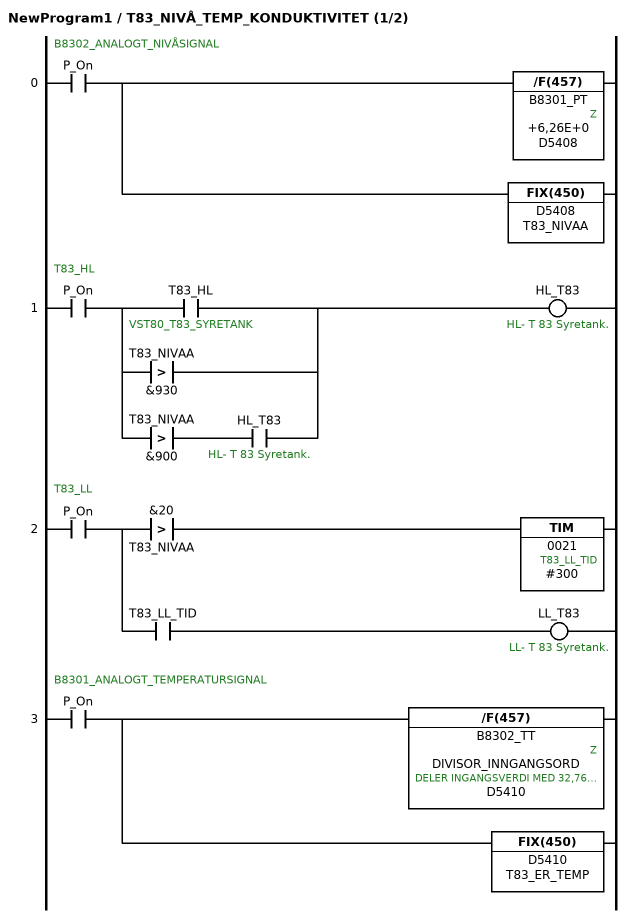
; [picture p48: NewProgram1 / T83_NIVÅ_TEMP_KONDUKTIVITET, rungs 0-3]
; rung 0: B8302_ANALOGT_NIVÅSIGNAL
LD P_On
/F(457) B8301_PT +6,26E+0 D5408  ; Z
FIX(450) D5408 T83_NIVAA
; rung 1: T83_HL
LD P_On
LD T83_HL  ; VST80_T83_SYRETANK
OR>(320) T83_NIVAA &930
LD>(320) T83_NIVAA &900
AND HL_T83  ; HL- T 83 Syretank.
ORLD
ANDLD
OUT HL_T83  ; HL- T 83 Syretank.
; rung 2: T83_LL
LD P_On
OUT TR0
AND>(320) &20 T83_NIVAA
TIM 0021 #300  ; T83_LL_TID
LD TR0
AND T83_LL_TID
OUT LL_T83  ; LL- T 83 Syretank.
; rung 3: B8301_ANALOGT_TEMPERATURSIGNAL
LD P_On
/F(457) B8302_TT DIVISOR_INNGANGSORD D5410  ; Z, DELER INGANGSVERDI MED 32,760 FOR OMREGNING TIL 0-1000
FIX(450) D5410 T83_ER_TEMP

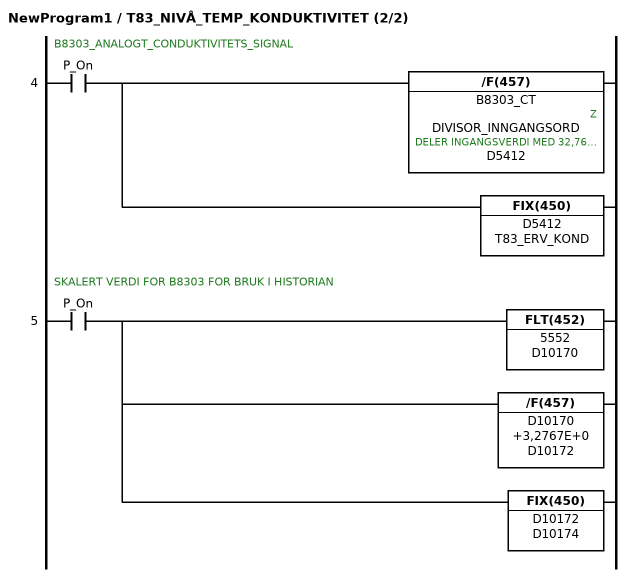
; rung 4: B8303_ANALOGT_CONDUKTIVITETS_SIGNAL
LD P_On
/F(457) B8303_CT DIVISOR_INNGANGSORD D5412  ; Z, DELER INGANGSVERDI MED 32,760 FOR OMREGNING TIL 0-1000
FIX(450) D5412 T83_ERV_KOND
; rung 5: SKALERT VERDI FOR B8303 FOR BRUK I HISTORIAN
LD P_On
FLT(452) 5552 D10170
/F(457) D10170 +3,2767E+0 D10172
FIX(450) D10172 D10174

### Section T83_FUNKSJONER_OBJEKTER

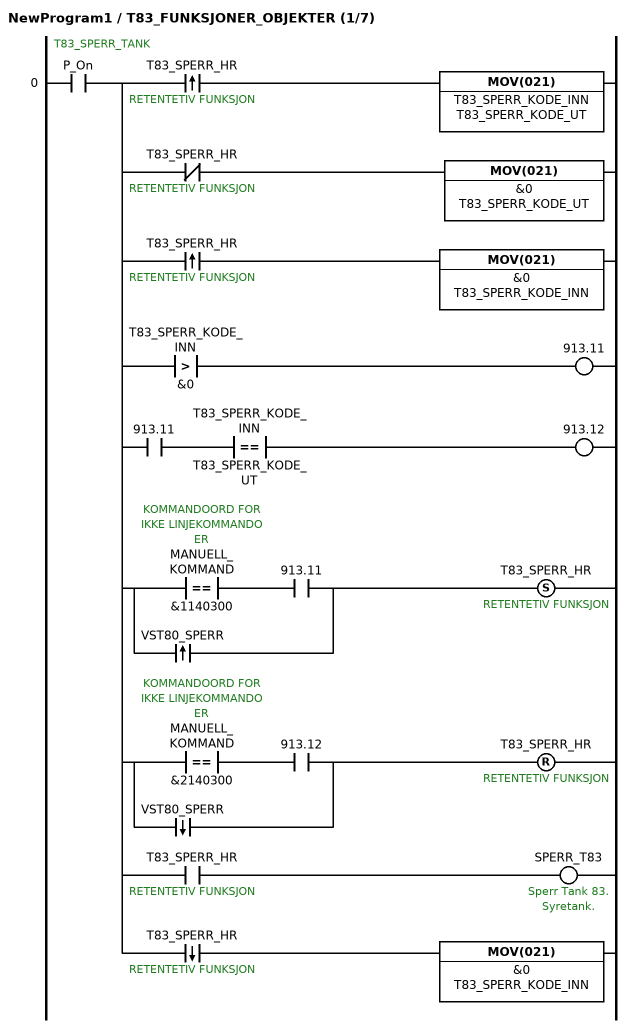
; rung 0: T83_SPERR_TANK
LD P_On
OUT TR0
@AND T83_SPERR_HR  ; RETENTETIV FUNKSJON
MOV(021) T83_SPERR_KODE_INN T83_SPERR_KODE_UT
LD TR0
ANDNOT T83_SPERR_HR  ; RETENTETIV FUNKSJON
MOV(021) &0 T83_SPERR_KODE_UT
LD TR0
@AND T83_SPERR_HR  ; RETENTETIV FUNKSJON
MOV(021) &0 T83_SPERR_KODE_INN
LD TR0
AND>(320) T83_SPERR_KODE_INN &0
OUT 913.11
LD TR0
AND 913.11
AND=(300) T83_SPERR_KODE_INN T83_SPERR_KODE_UT
OUT 913.12
LD TR0
LD=L(301) MANUELL_KOMMAND &1140300  ; KOMMANDOORD FOR IKKE LINJEKOMMANDOER
AND 913.11
@OR VST80_SPERR
ANDLD
SET T83_SPERR_HR  ; RETENTETIV FUNKSJON
LD TR0
LD=L(301) MANUELL_KOMMAND &2140300  ; KOMMANDOORD FOR IKKE LINJEKOMMANDOER
AND 913.12
%OR VST80_SPERR
ANDLD
RSET T83_SPERR_HR  ; RETENTETIV FUNKSJON
LD TR0
AND T83_SPERR_HR  ; RETENTETIV FUNKSJON
OUT SPERR_T83  ; Sperr Tank 83. Syretank.
LD TR0
%AND T83_SPERR_HR  ; RETENTETIV FUNKSJON
MOV(021) &0 T83_SPERR_KODE_INN

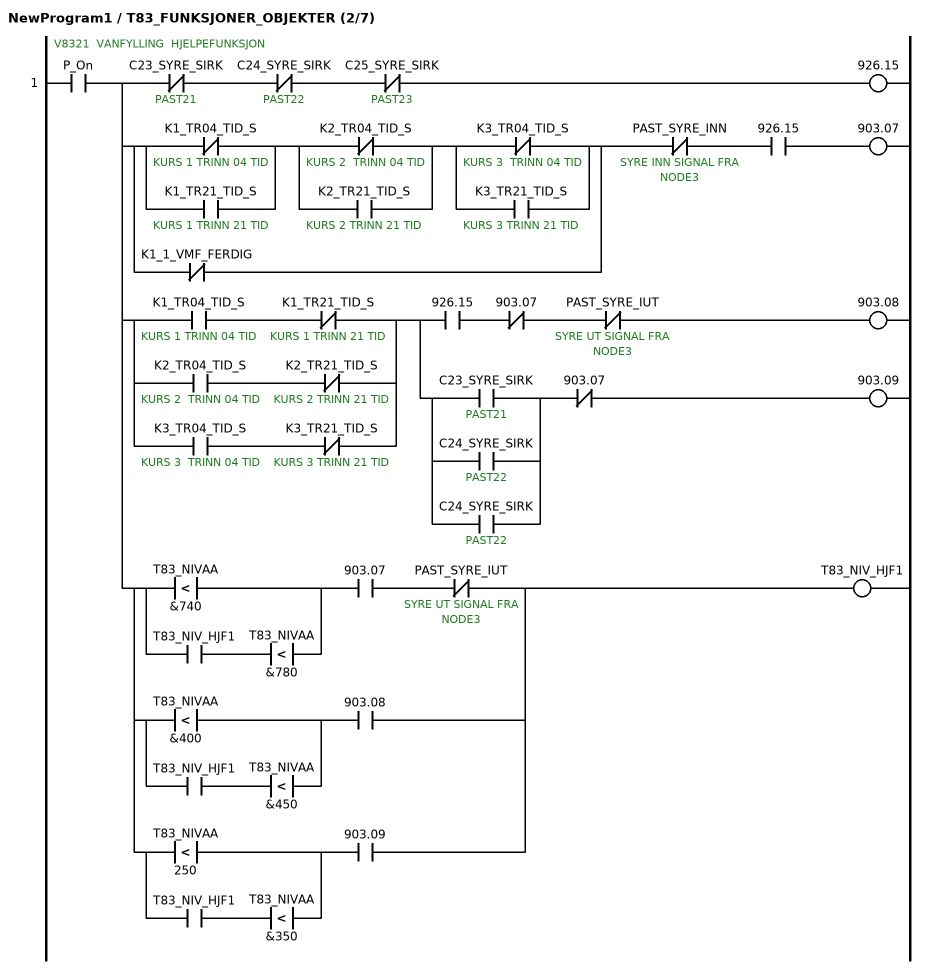
; rung 1: V8321  VANFYLLING  HJELPEFUNKSJON
LD P_On
OUT TR0
ANDNOT C23_SYRE_SIRK  ; PAST21
ANDNOT C24_SYRE_SIRK  ; PAST22
ANDNOT C25_SYRE_SIRK  ; PAST23
OUT 926.15
LD TR0
LDNOT K1_TR04_TID_S  ; KURS 1 TRINN 04 TID
OR K1_TR21_TID_S  ; KURS 1 TRINN 21 TID
LDNOT K2_TR04_TID_S  ; KURS 2  TRINN 04 TID
OR K2_TR21_TID_S  ; KURS 2 TRINN 21 TID
ANDLD
LDNOT K3_TR04_TID_S  ; KURS 3  TRINN 04 TID
OR K3_TR21_TID_S  ; KURS 3 TRINN 21 TID
ANDLD
ORNOT K1_1_VMF_FERDIG
ANDLD
ANDNOT PAST_SYRE_INN  ; SYRE INN SIGNAL FRA NODE3
AND 926.15
OUT 903.07
LD TR0
LD K1_TR04_TID_S  ; KURS 1 TRINN 04 TID
ANDNOT K1_TR21_TID_S  ; KURS 1 TRINN 21 TID
LD K2_TR04_TID_S  ; KURS 2  TRINN 04 TID
ANDNOT K2_TR21_TID_S  ; KURS 2 TRINN 21 TID
ORLD
LD K3_TR04_TID_S  ; KURS 3  TRINN 04 TID
ANDNOT K3_TR21_TID_S  ; KURS 3 TRINN 21 TID
ORLD
ANDLD
OUT TR1
AND 926.15
ANDNOT 903.07
ANDNOT PAST_SYRE_IUT  ; SYRE UT SIGNAL FRA NODE3
OUT 903.08
LD TR1
LD C23_SYRE_SIRK  ; PAST21
OR C24_SYRE_SIRK  ; PAST22
OR C24_SYRE_SIRK  ; PAST22
ANDLD
ANDNOT 903.07
OUT 903.09
LD TR0
LD<(310) T83_NIVAA &740
LD T83_NIV_HJF1
AND<(310) T83_NIVAA &780
ORLD
AND 903.07
ANDNOT PAST_SYRE_IUT  ; SYRE UT SIGNAL FRA NODE3
LD<(310) T83_NIVAA &400
LD T83_NIV_HJF1
AND<(310) T83_NIVAA &450
ORLD
AND 903.08
ORLD
LD<(310) T83_NIVAA 250
LD T83_NIV_HJF1
AND<(310) T83_NIVAA &350
ORLD
AND 903.09
ORLD
ANDLD
OUT T83_NIV_HJF1

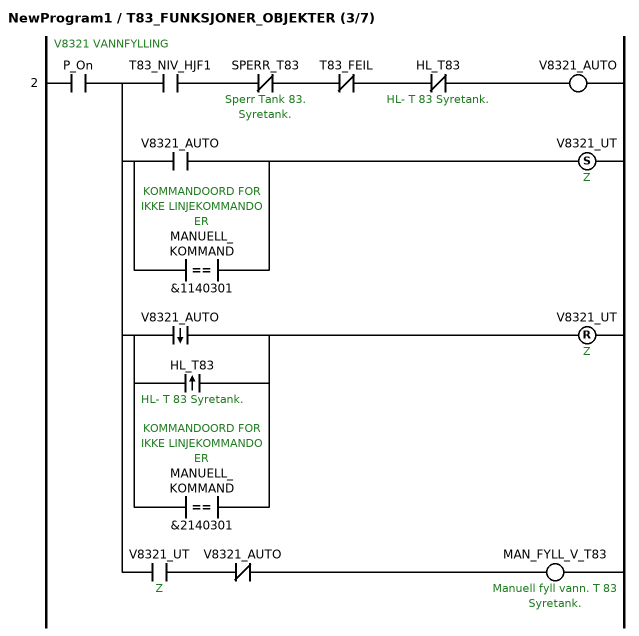
; rung 2: V8321 VANNFYLLING
LD P_On
OUT TR0
AND T83_NIV_HJF1
ANDNOT SPERR_T83  ; Sperr Tank 83. Syretank.
ANDNOT T83_FEIL
ANDNOT HL_T83  ; HL- T 83 Syretank.
OUT V8321_AUTO
LD TR0
LD V8321_AUTO
OR=L(301) MANUELL_KOMMAND &1140301  ; KOMMANDOORD FOR IKKE LINJEKOMMANDOER
ANDLD
SET V8321_UT  ; Z
LD TR0
%LD V8321_AUTO
@OR HL_T83  ; HL- T 83 Syretank.
OR=L(301) MANUELL_KOMMAND &2140301  ; KOMMANDOORD FOR IKKE LINJEKOMMANDOER
ANDLD
RSET V8321_UT  ; Z
LD TR0
AND V8321_UT  ; Z
ANDNOT V8321_AUTO
OUT MAN_FYLL_V_T83  ; Manuell fyll vann. T 83 Syretank.

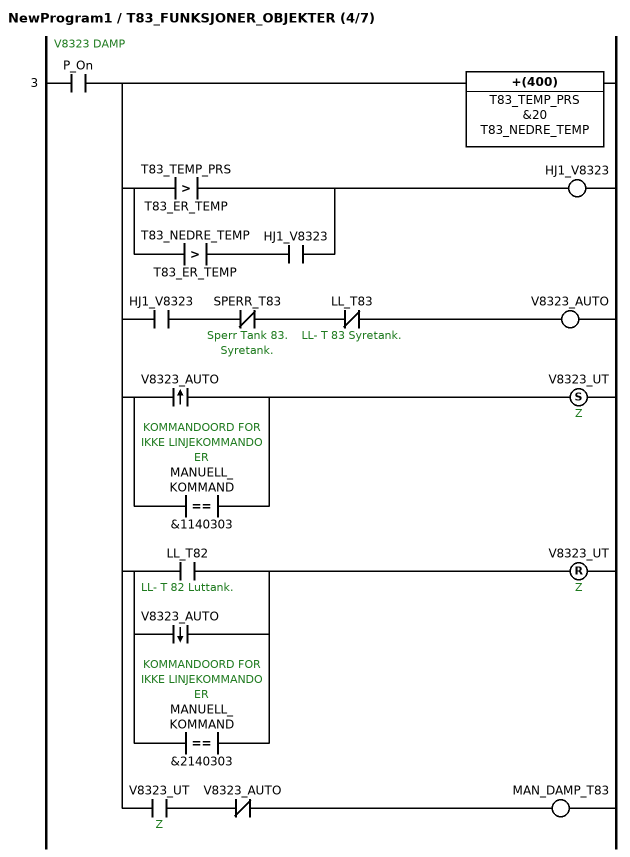
; rung 3: V8323 DAMP
LD P_On
OUT TR0
+(400) T83_TEMP_PRS &20 T83_NEDRE_TEMP
LD>(320) T83_TEMP_PRS T83_ER_TEMP
LD>(320) T83_NEDRE_TEMP T83_ER_TEMP
AND HJ1_V8323
ORLD
ANDLD
OUT HJ1_V8323
LD TR0
AND HJ1_V8323
ANDNOT SPERR_T83  ; Sperr Tank 83. Syretank.
ANDNOT LL_T83  ; LL- T 83 Syretank.
OUT V8323_AUTO
LD TR0
@LD V8323_AUTO
OR=L(301) MANUELL_KOMMAND &1140303  ; KOMMANDOORD FOR IKKE LINJEKOMMANDOER
ANDLD
SET V8323_UT  ; Z
LD TR0
LD LL_T82  ; LL- T 82 Luttank.
%OR V8323_AUTO
OR=L(301) MANUELL_KOMMAND &2140303  ; KOMMANDOORD FOR IKKE LINJEKOMMANDOER
ANDLD
RSET V8323_UT  ; Z
LD TR0
AND V8323_UT  ; Z
ANDNOT V8323_AUTO
OUT MAN_DAMP_T83

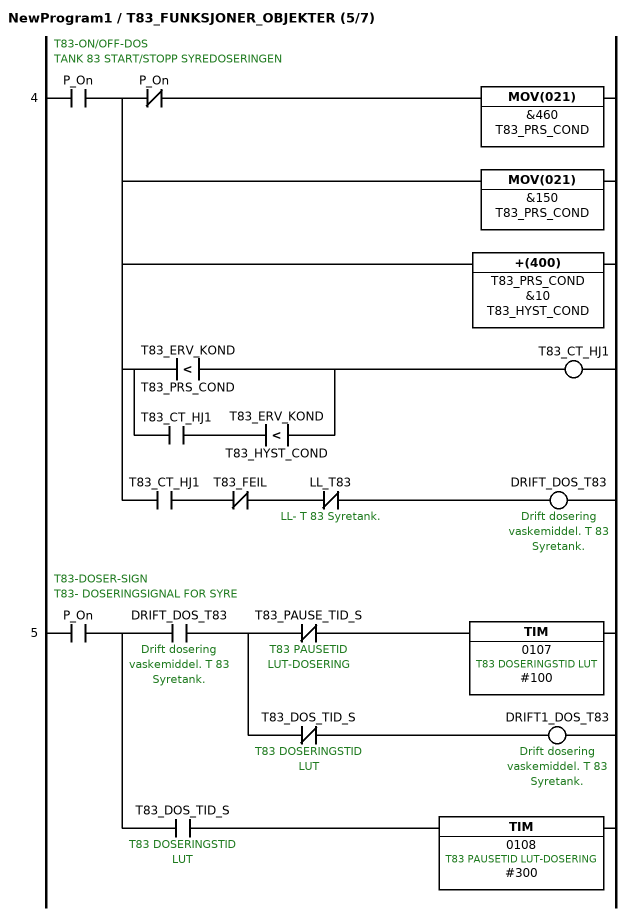
; rung 4: T83-ON/OFF-DOS / TANK 83 START/STOPP SYREDOSERINGEN
LD P_On
OUT TR0
ANDNOT P_On
MOV(021) &460 T83_PRS_COND
LD TR0
MOV(021) &150 T83_PRS_COND
+(400) T83_PRS_COND &10 T83_HYST_COND
LD<(310) T83_ERV_KOND T83_PRS_COND
LD T83_CT_HJ1
AND<(310) T83_ERV_KOND T83_HYST_COND
ORLD
ANDLD
OUT T83_CT_HJ1
LD TR0
AND T83_CT_HJ1
ANDNOT T83_FEIL
ANDNOT LL_T83  ; LL- T 83 Syretank.
OUT DRIFT_DOS_T83  ; Drift dosering vaskemiddel. T 83 Syretank.
; rung 5: T83-DOSER-SIGN / T83- DOSERINGSIGNAL FOR SYRE
LD P_On
OUT TR0
AND DRIFT_DOS_T83  ; Drift dosering vaskemiddel. T 83 Syretank.
OUT TR1
ANDNOT T83_PAUSE_TID_S  ; T83 PAUSETID LUT-DOSERING
TIM 0107 #100  ; T83 DOSERINGSTID LUT
LD TR1
ANDNOT T83_DOS_TID_S  ; T83 DOSERINGSTID LUT
OUT DRIFT1_DOS_T83  ; Drift dosering vaskemiddel. T 83 Syretank.
LD TR0
AND T83_DOS_TID_S  ; T83 DOSERINGSTID LUT
TIM 0108 #300  ; T83 PAUSETID LUT-DOSERING

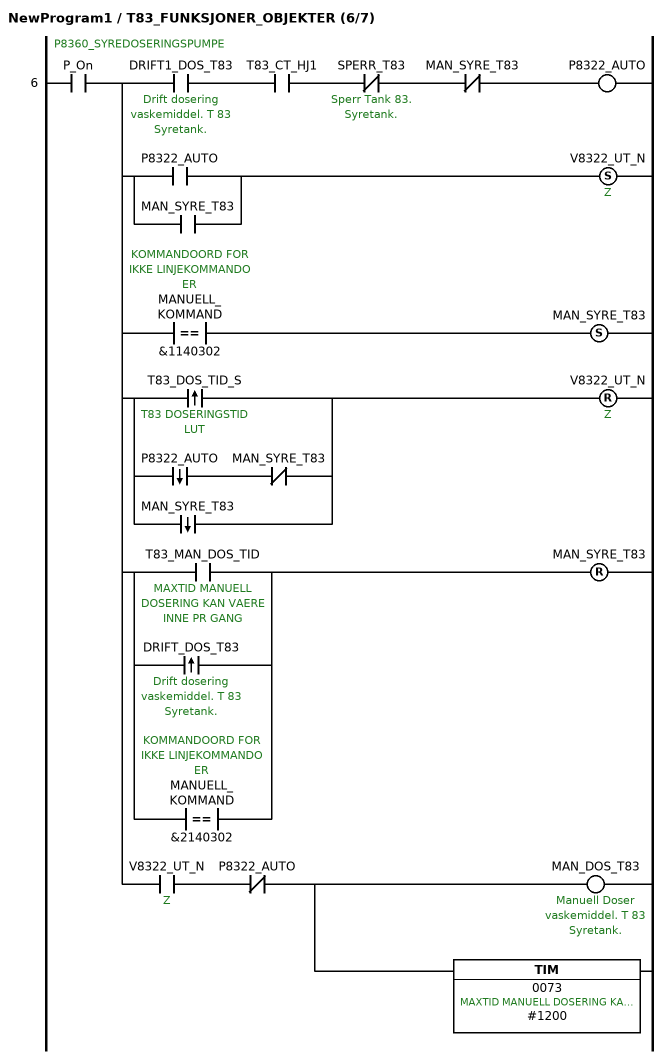
; rung 6: P8360_SYREDOSERINGSPUMPE
LD P_On
OUT TR0
AND DRIFT1_DOS_T83  ; Drift dosering vaskemiddel. T 83 Syretank.
AND T83_CT_HJ1
ANDNOT SPERR_T83  ; Sperr Tank 83. Syretank.
ANDNOT MAN_SYRE_T83
OUT P8322_AUTO
LD TR0
LD P8322_AUTO
OR MAN_SYRE_T83
ANDLD
SET V8322_UT_N  ; Z
LD TR0
AND=L(301) MANUELL_KOMMAND &1140302  ; KOMMANDOORD FOR IKKE LINJEKOMMANDOER
SET MAN_SYRE_T83
LD TR0
@LD T83_DOS_TID_S  ; T83 DOSERINGSTID LUT
%LD P8322_AUTO
ANDNOT MAN_SYRE_T83
ORLD
%OR MAN_SYRE_T83
ANDLD
RSET V8322_UT_N  ; Z
LD TR0
LD T83_MAN_DOS_TID  ; MAXTID MANUELL DOSERING KAN VAERE INNE PR GANG
@OR DRIFT_DOS_T83  ; Drift dosering vaskemiddel. T 83 Syretank.
OR=L(301) MANUELL_KOMMAND &2140302  ; KOMMANDOORD FOR IKKE LINJEKOMMANDOER
ANDLD
RSET MAN_SYRE_T83
LD TR0
AND V8322_UT_N  ; Z
ANDNOT P8322_AUTO
OUT MAN_DOS_T83  ; Manuell Doser vaskemiddel. T 83 Syretank.
TIM 0073 #1200  ; MAXTID MANUELL DOSERING KAN VAERE INNE PR GANG

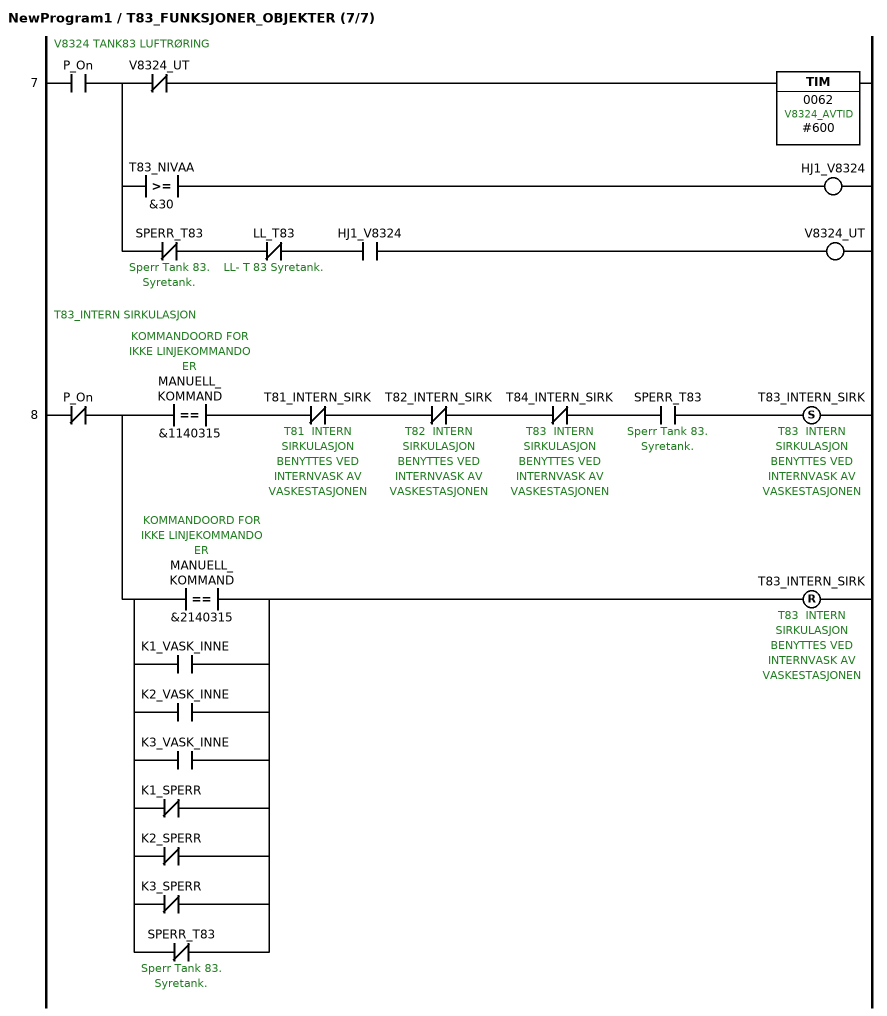
; rung 7: V8324 TANK83 LUFTRØRING
LD P_On
OUT TR0
ANDNOT V8324_UT
TIM 0062 #600  ; V8324_AVTID
LD TR0
AND>=(325) T83_NIVAA &30
OUT HJ1_V8324
LD TR0
ANDNOT SPERR_T83  ; Sperr Tank 83. Syretank.
ANDNOT LL_T83  ; LL- T 83 Syretank.
AND HJ1_V8324
OUT V8324_UT
; rung 8: T83_INTERN SIRKULASJON
LDNOT P_On
OUT TR0
AND=L(301) MANUELL_KOMMAND &1140315  ; KOMMANDOORD FOR IKKE LINJEKOMMANDOER
ANDNOT T81_INTERN_SIRK  ; T81  INTERN SIRKULASJON BENYTTES VED INTERNVASK AV VASKESTASJONEN
ANDNOT T82_INTERN_SIRK  ; T82  INTERN SIRKULASJON BENYTTES VED INTERNVASK AV VASKESTASJONEN
ANDNOT T84_INTERN_SIRK  ; T83  INTERN SIRKULASJON BENYTTES VED INTERNVASK AV VASKESTASJONEN
AND SPERR_T83  ; Sperr Tank 83. Syretank.
SET T83_INTERN_SIRK  ; T83  INTERN SIRKULASJON BENYTTES VED INTERNVASK AV VASKESTASJONEN
LD TR0
LD=L(301) MANUELL_KOMMAND &2140315  ; KOMMANDOORD FOR IKKE LINJEKOMMANDOER
OR K1_VASK_INNE
OR K2_VASK_INNE
OR K3_VASK_INNE
ORNOT K1_SPERR
ORNOT K2_SPERR
ORNOT K3_SPERR
ORNOT SPERR_T83  ; Sperr Tank 83. Syretank.
ANDLD
RSET T83_INTERN_SIRK  ; T83  INTERN SIRKULASJON BENYTTES VED INTERNVASK AV VASKESTASJONEN

### Section T84_NIVÅ_TEMPERATUR_CONDUKTIVITET

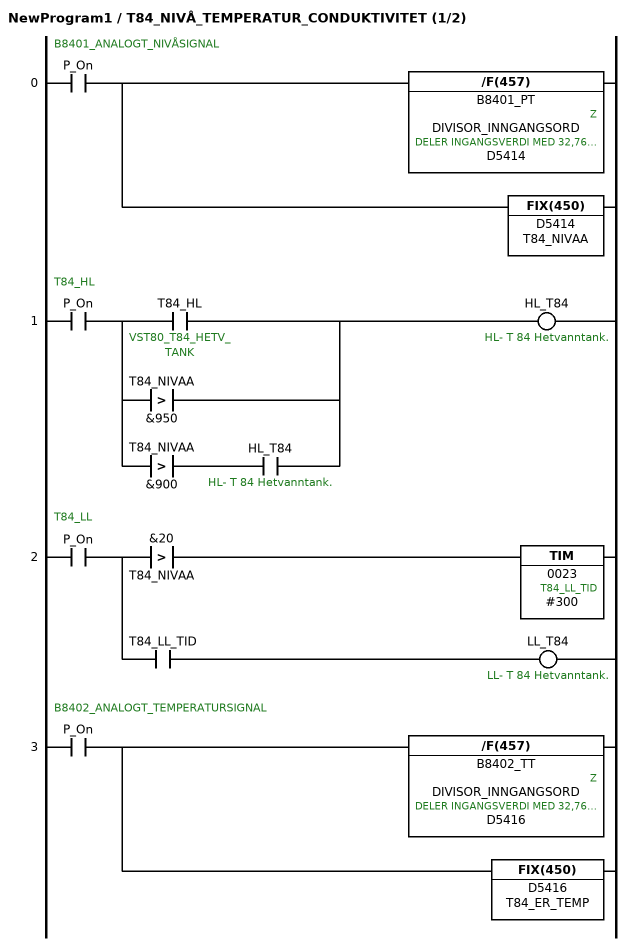
; rung 0: B8401_ANALOGT_NIVÅSIGNAL
LD P_On
/F(457) B8401_PT DIVISOR_INNGANGSORD D5414  ; Z, DELER INGANGSVERDI MED 32,760 FOR OMREGNING TIL 0-1000
FIX(450) D5414 T84_NIVAA
; rung 1: T84_HL
LD P_On
LD T84_HL  ; VST80_T84_HETV_TANK
OR>(320) T84_NIVAA &950
LD>(320) T84_NIVAA &900
AND HL_T84  ; HL- T 84 Hetvanntank.
ORLD
ANDLD
OUT HL_T84  ; HL- T 84 Hetvanntank.
; rung 2: T84_LL
LD P_On
OUT TR0
AND>(320) &20 T84_NIVAA
TIM 0023 #300  ; T84_LL_TID
LD TR0
AND T84_LL_TID
OUT LL_T84  ; LL- T 84 Hetvanntank.
; rung 3: B8402_ANALOGT_TEMPERATURSIGNAL
LD P_On
/F(457) B8402_TT DIVISOR_INNGANGSORD D5416  ; Z, DELER INGANGSVERDI MED 32,760 FOR OMREGNING TIL 0-1000
FIX(450) D5416 T84_ER_TEMP

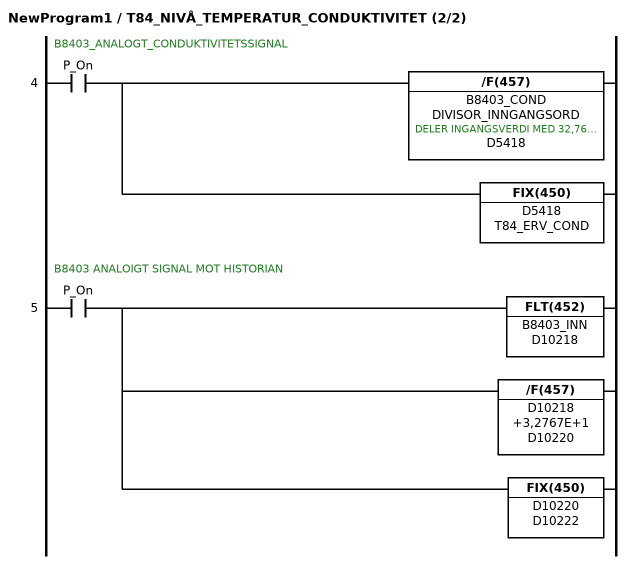
; rung 4: B8403_ANALOGT_CONDUKTIVITETSSIGNAL
LD P_On
/F(457) B8403_COND DIVISOR_INNGANGSORD D5418  ; DELER INGANGSVERDI MED 32,760 FOR OMREGNING TIL 0-1000
FIX(450) D5418 T84_ERV_COND
; rung 5: B8403 ANALOIGT SIGNAL MOT HISTORIAN
LD P_On
FLT(452) B8403_INN D10218
/F(457) D10218 +3,2767E+1 D10220
FIX(450) D10220 D10222

### Section T84_FUNKSJONER_OBJEKTER

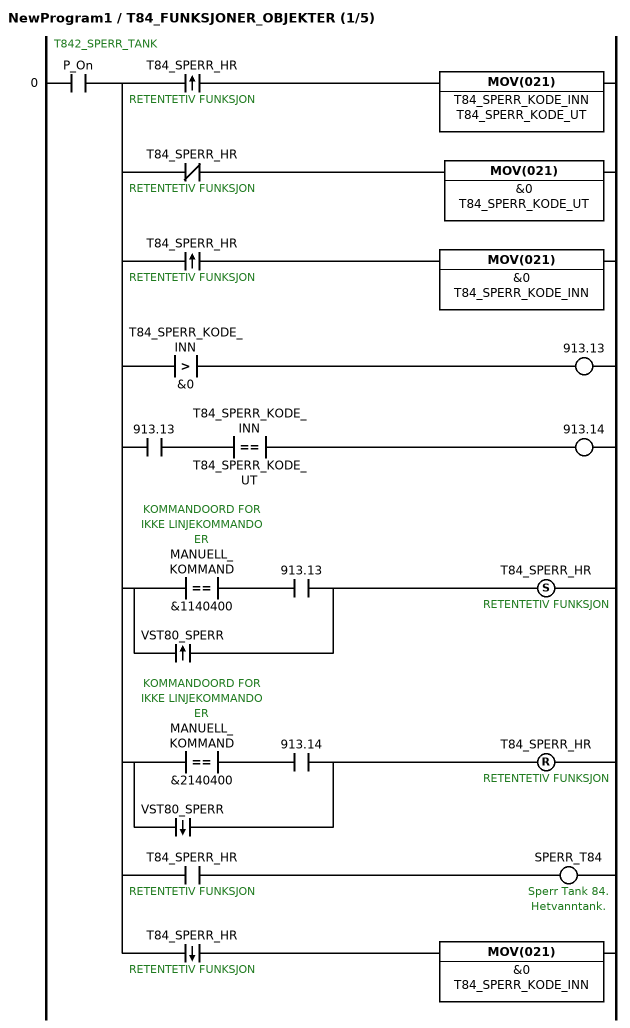
; rung 0: T842_SPERR_TANK
LD P_On
OUT TR0
@AND T84_SPERR_HR  ; RETENTETIV FUNKSJON
MOV(021) T84_SPERR_KODE_INN T84_SPERR_KODE_UT
LD TR0
ANDNOT T84_SPERR_HR  ; RETENTETIV FUNKSJON
MOV(021) &0 T84_SPERR_KODE_UT
LD TR0
@AND T84_SPERR_HR  ; RETENTETIV FUNKSJON
MOV(021) &0 T84_SPERR_KODE_INN
LD TR0
AND>(320) T84_SPERR_KODE_INN &0
OUT 913.13
LD TR0
AND 913.13
AND=(300) T84_SPERR_KODE_INN T84_SPERR_KODE_UT
OUT 913.14
LD TR0
LD=L(301) MANUELL_KOMMAND &1140400  ; KOMMANDOORD FOR IKKE LINJEKOMMANDOER
AND 913.13
@OR VST80_SPERR
ANDLD
SET T84_SPERR_HR  ; RETENTETIV FUNKSJON
LD TR0
LD=L(301) MANUELL_KOMMAND &2140400  ; KOMMANDOORD FOR IKKE LINJEKOMMANDOER
AND 913.14
%OR VST80_SPERR
ANDLD
RSET T84_SPERR_HR  ; RETENTETIV FUNKSJON
LD TR0
AND T84_SPERR_HR  ; RETENTETIV FUNKSJON
OUT SPERR_T84  ; Sperr Tank 84. Hetvanntank.
LD TR0
%AND T84_SPERR_HR  ; RETENTETIV FUNKSJON
MOV(021) &0 T84_SPERR_KODE_INN

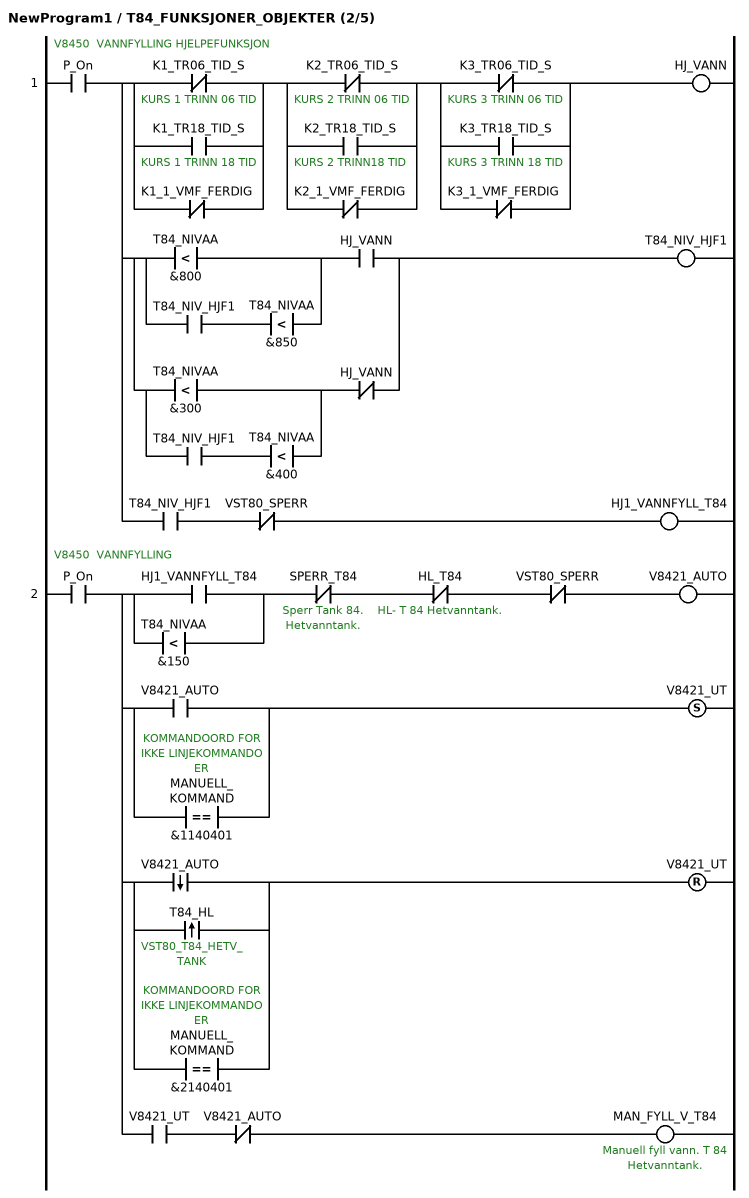
; rung 1: V8450  VANNFYLLING HJELPEFUNKSJON
LD P_On
OUT TR0
LDNOT K1_TR06_TID_S  ; KURS 1 TRINN 06 TID
OR K1_TR18_TID_S  ; KURS 1 TRINN 18 TID
ORNOT K1_1_VMF_FERDIG
ANDLD
LDNOT K2_TR06_TID_S  ; KURS 2 TRINN 06 TID
OR K2_TR18_TID_S  ; KURS 2 TRINN18 TID
ORNOT K2_1_VMF_FERDIG
ANDLD
LDNOT K3_TR06_TID_S  ; KURS 3 TRINN 06 TID
OR K3_TR18_TID_S  ; KURS 3 TRINN 18 TID
ORNOT K3_1_VMF_FERDIG
ANDLD
OUT HJ_VANN
LD TR0
LD<(310) T84_NIVAA &800
LD T84_NIV_HJF1
AND<(310) T84_NIVAA &850
ORLD
AND HJ_VANN
LD<(310) T84_NIVAA &300
LD T84_NIV_HJF1
AND<(310) T84_NIVAA &400
ORLD
ANDNOT HJ_VANN
ORLD
ANDLD
OUT T84_NIV_HJF1
LD TR0
AND T84_NIV_HJF1
ANDNOT VST80_SPERR
OUT HJ1_VANNFYLL_T84
; rung 2: V8450  VANNFYLLING
LD P_On
OUT TR0
LD HJ1_VANNFYLL_T84
OR<(310) T84_NIVAA &150
ANDLD
ANDNOT SPERR_T84  ; Sperr Tank 84. Hetvanntank.
ANDNOT HL_T84  ; HL- T 84 Hetvanntank.
ANDNOT VST80_SPERR
OUT V8421_AUTO
LD TR0
LD V8421_AUTO
OR=L(301) MANUELL_KOMMAND &1140401  ; KOMMANDOORD FOR IKKE LINJEKOMMANDOER
ANDLD
SET V8421_UT
LD TR0
%LD V8421_AUTO
@OR T84_HL  ; VST80_T84_HETV_TANK
OR=L(301) MANUELL_KOMMAND &2140401  ; KOMMANDOORD FOR IKKE LINJEKOMMANDOER
ANDLD
RSET V8421_UT
LD TR0
AND V8421_UT
ANDNOT V8421_AUTO
OUT MAN_FYLL_V_T84  ; Manuell fyll vann. T 84 Hetvanntank.

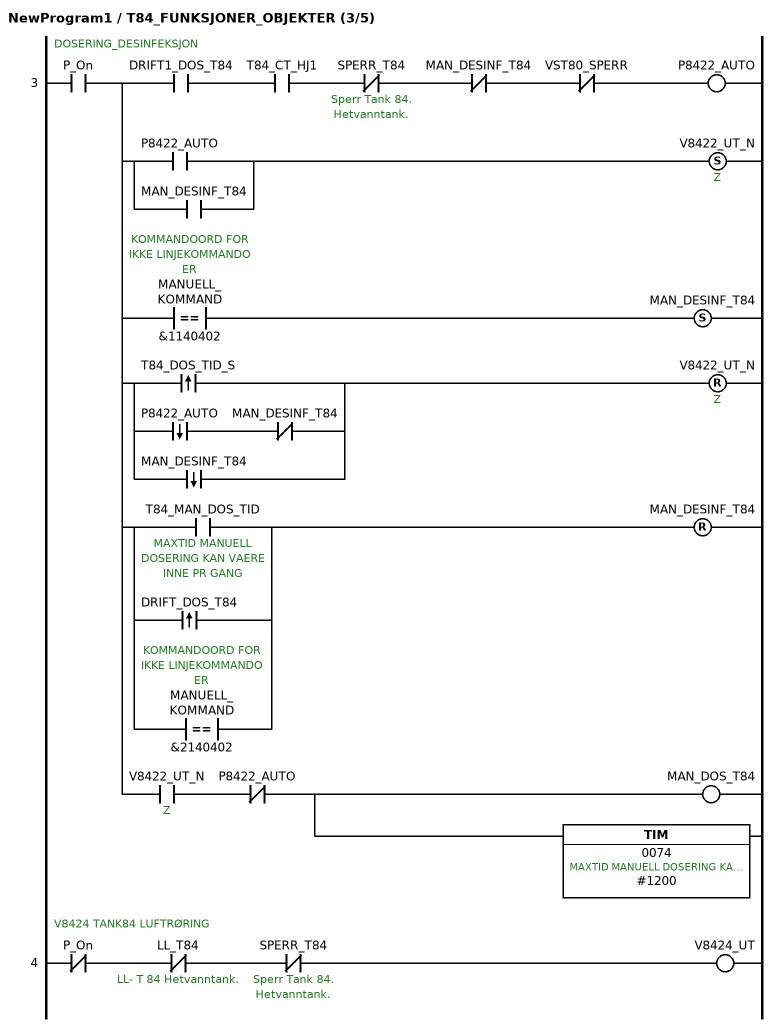
; rung 3: DOSERING_DESINFEKSJON
LD P_On
OUT TR0
AND DRIFT1_DOS_T84
AND T84_CT_HJ1
ANDNOT SPERR_T84  ; Sperr Tank 84. Hetvanntank.
ANDNOT MAN_DESINF_T84
ANDNOT VST80_SPERR
OUT P8422_AUTO
LD TR0
LD P8422_AUTO
OR MAN_DESINF_T84
ANDLD
SET V8422_UT_N  ; Z
LD TR0
AND=L(301) MANUELL_KOMMAND &1140402  ; KOMMANDOORD FOR IKKE LINJEKOMMANDOER
SET MAN_DESINF_T84
LD TR0
@LD T84_DOS_TID_S
%LD P8422_AUTO
ANDNOT MAN_DESINF_T84
ORLD
%OR MAN_DESINF_T84
ANDLD
RSET V8422_UT_N  ; Z
LD TR0
LD T84_MAN_DOS_TID  ; MAXTID MANUELL DOSERING KAN VAERE INNE PR GANG
@OR DRIFT_DOS_T84
OR=L(301) MANUELL_KOMMAND &2140402  ; KOMMANDOORD FOR IKKE LINJEKOMMANDOER
ANDLD
RSET MAN_DESINF_T84
LD TR0
AND V8422_UT_N  ; Z
ANDNOT P8422_AUTO
OUT MAN_DOS_T84
TIM 0074 #1200  ; MAXTID MANUELL DOSERING KAN VAERE INNE PR GANG
; rung 4: V8424 TANK84 LUFTRØRING
LDNOT P_On
ANDNOT LL_T84  ; LL- T 84 Hetvanntank.
ANDNOT SPERR_T84  ; Sperr Tank 84. Hetvanntank.
OUT V8424_UT

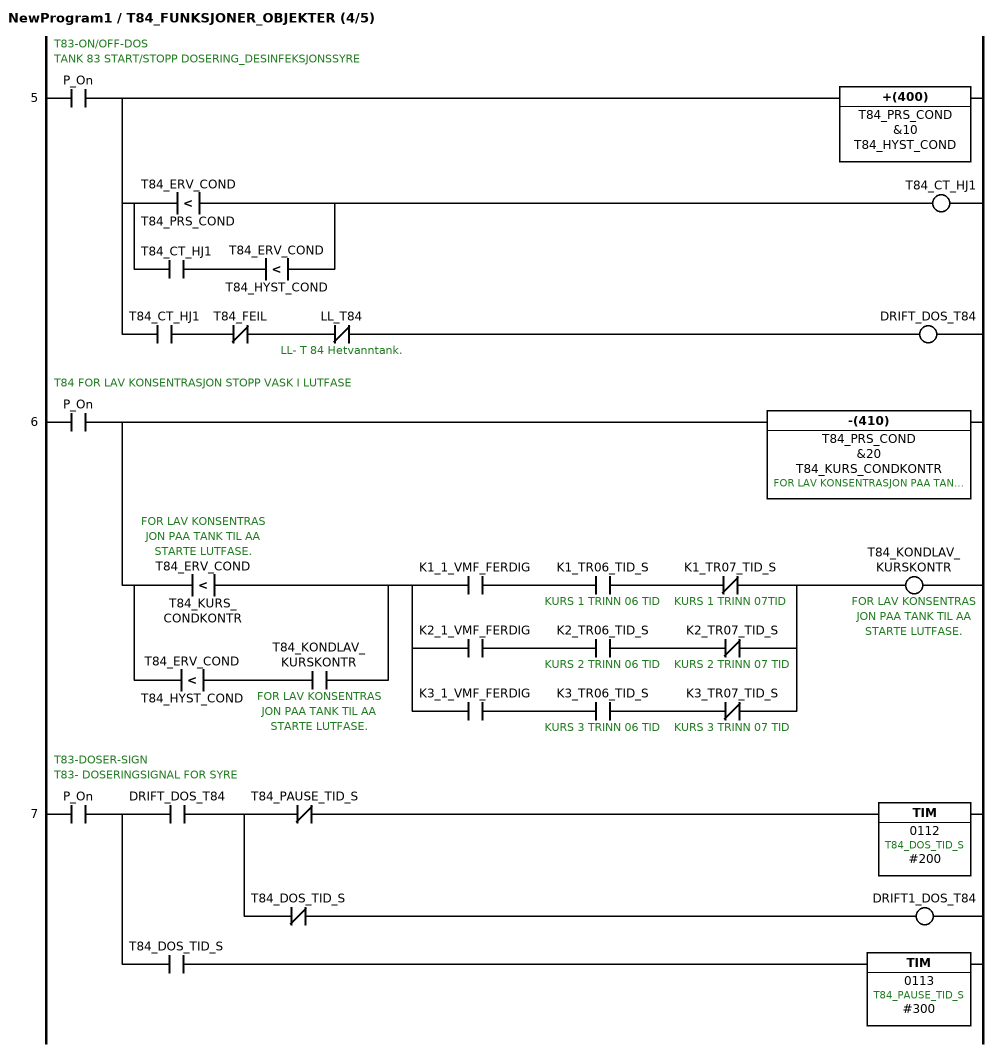
; rung 5: T83-ON/OFF-DOS / TANK 83 START/STOPP DOSERING_DESINFEKSJONSSYRE
LD P_On
OUT TR0
+(400) T84_PRS_COND &10 T84_HYST_COND
LD<(310) T84_ERV_COND T84_PRS_COND
LD T84_CT_HJ1
AND<(310) T84_ERV_COND T84_HYST_COND
ORLD
ANDLD
OUT T84_CT_HJ1
LD TR0
AND T84_CT_HJ1
ANDNOT T84_FEIL
ANDNOT LL_T84  ; LL- T 84 Hetvanntank.
OUT DRIFT_DOS_T84
; rung 6: T84 FOR LAV KONSENTRASJON STOPP VASK I LUTFASE
LD P_On
-(410) T84_PRS_COND &20 T84_KURS_CONDKONTR  ; FOR LAV KONSENTRASJON PAA TANK TIL AA STARTE LUTFASE.
LD<(310) T84_ERV_COND T84_KURS_CONDKONTR  ; FOR LAV KONSENTRASJON PAA TANK TIL AA STARTE LUTFASE.
LD<(310) T84_ERV_COND T84_HYST_COND
AND T84_KONDLAV_KURSKONTR  ; FOR LAV KONSENTRASJON PAA TANK TIL AA STARTE LUTFASE.
ORLD
ANDLD
LD K1_1_VMF_FERDIG
AND K1_TR06_TID_S  ; KURS 1 TRINN 06 TID
ANDNOT K1_TR07_TID_S  ; KURS 1 TRINN 07TID
LD K2_1_VMF_FERDIG
AND K2_TR06_TID_S  ; KURS 2 TRINN 06 TID
ANDNOT K2_TR07_TID_S  ; KURS 2 TRINN 07 TID
ORLD
LD K3_1_VMF_FERDIG
AND K3_TR06_TID_S  ; KURS 3 TRINN 06 TID
ANDNOT K3_TR07_TID_S  ; KURS 3 TRINN 07 TID
ORLD
ANDLD
OUT T84_KONDLAV_KURSKONTR  ; FOR LAV KONSENTRASJON PAA TANK TIL AA STARTE LUTFASE.
; rung 7: T83-DOSER-SIGN / T83- DOSERINGSIGNAL FOR SYRE
LD P_On
OUT TR0
AND DRIFT_DOS_T84
OUT TR1
ANDNOT T84_PAUSE_TID_S
TIM 0112 #200  ; T84_DOS_TID_S
LD TR1
ANDNOT T84_DOS_TID_S
OUT DRIFT1_DOS_T84
LD TR0
AND T84_DOS_TID_S
TIM 0113 #300  ; T84_PAUSE_TID_S

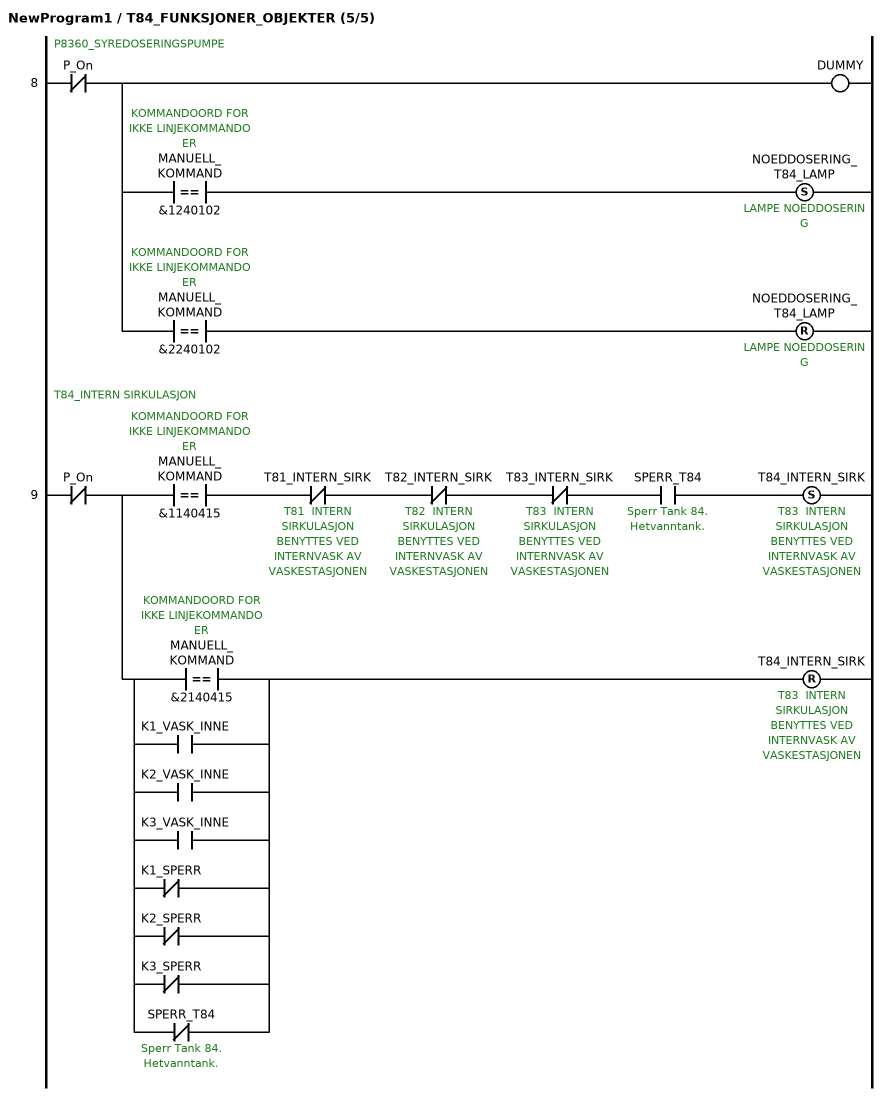
; rung 8: P8360_SYREDOSERINGSPUMPE
LDNOT P_On
OUT TR0
OUT DUMMY
AND=L(301) MANUELL_KOMMAND &1240102  ; KOMMANDOORD FOR IKKE LINJEKOMMANDOER
SET NOEDDOSERING_T84_LAMP  ; LAMPE NOEDDOSERING
LD TR0
AND=L(301) MANUELL_KOMMAND &2240102  ; KOMMANDOORD FOR IKKE LINJEKOMMANDOER
RSET NOEDDOSERING_T84_LAMP  ; LAMPE NOEDDOSERING
; rung 9: T84_INTERN SIRKULASJON
LDNOT P_On
OUT TR0
AND=L(301) MANUELL_KOMMAND &1140415  ; KOMMANDOORD FOR IKKE LINJEKOMMANDOER
ANDNOT T81_INTERN_SIRK  ; T81  INTERN SIRKULASJON BENYTTES VED INTERNVASK AV VASKESTASJONEN
ANDNOT T82_INTERN_SIRK  ; T82  INTERN SIRKULASJON BENYTTES VED INTERNVASK AV VASKESTASJONEN
ANDNOT T83_INTERN_SIRK  ; T83  INTERN SIRKULASJON BENYTTES VED INTERNVASK AV VASKESTASJONEN
AND SPERR_T84  ; Sperr Tank 84. Hetvanntank.
SET T84_INTERN_SIRK  ; T83  INTERN SIRKULASJON BENYTTES VED INTERNVASK AV VASKESTASJONEN
LD TR0
LD=L(301) MANUELL_KOMMAND &2140415  ; KOMMANDOORD FOR IKKE LINJEKOMMANDOER
OR K1_VASK_INNE
OR K2_VASK_INNE
OR K3_VASK_INNE
ORNOT K1_SPERR
ORNOT K2_SPERR
ORNOT K3_SPERR
ORNOT SPERR_T84  ; Sperr Tank 84. Hetvanntank.
ANDLD
RSET T84_INTERN_SIRK  ; T83  INTERN SIRKULASJON BENYTTES VED INTERNVASK AV VASKESTASJONEN

### Section VST80_TANKFEIL

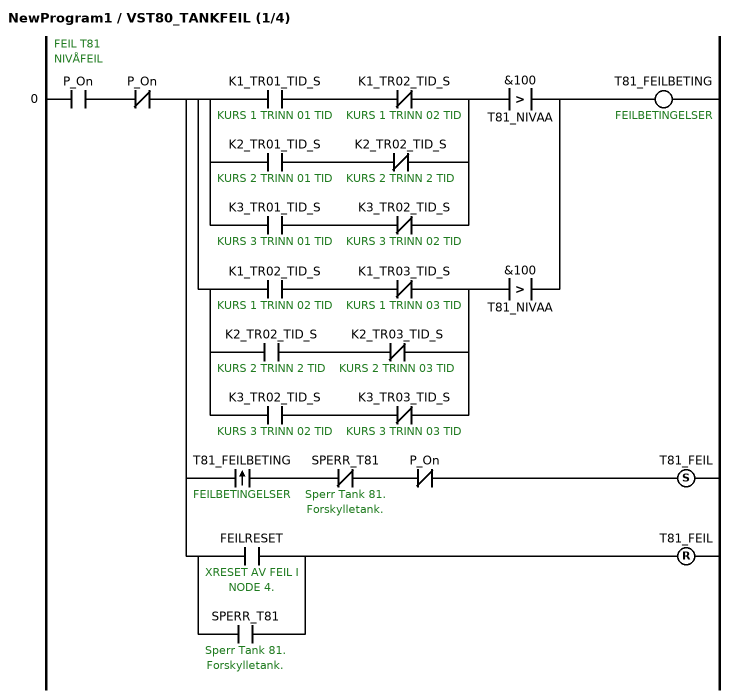
; rung 0: FEIL T81 / NIVÅFEIL
LD P_On
ANDNOT P_On
OUT TR0
LD K1_TR01_TID_S  ; KURS 1 TRINN 01 TID
ANDNOT K1_TR02_TID_S  ; KURS 1 TRINN 02 TID
LD K2_TR01_TID_S  ; KURS 2 TRINN 01 TID
ANDNOT K2_TR02_TID_S  ; KURS 2 TRINN 2 TID
ORLD
LD K3_TR01_TID_S  ; KURS 3 TRINN 01 TID
ANDNOT K3_TR02_TID_S  ; KURS 3 TRINN 02 TID
ORLD
AND>(320) &100 T81_NIVAA
LD K1_TR02_TID_S  ; KURS 1 TRINN 02 TID
ANDNOT K1_TR03_TID_S  ; KURS 1 TRINN 03 TID
LD K2_TR02_TID_S  ; KURS 2 TRINN 2 TID
ANDNOT K2_TR03_TID_S  ; KURS 2 TRINN 03 TID
ORLD
LD K3_TR02_TID_S  ; KURS 3 TRINN 02 TID
ANDNOT K3_TR03_TID_S  ; KURS 3 TRINN 03 TID
ORLD
AND>(320) &100 T81_NIVAA
ORLD
ANDLD
OUT T81_FEILBETING  ; FEILBETINGELSER
LD TR0
@AND T81_FEILBETING  ; FEILBETINGELSER
ANDNOT SPERR_T81  ; Sperr Tank 81. Forskylletank.
ANDNOT P_On
SET T81_FEIL
LD TR0
LD FEILRESET  ; XRESET AV FEIL I NODE 4.
OR SPERR_T81  ; Sperr Tank 81. Forskylletank.
ANDLD
RSET T81_FEIL

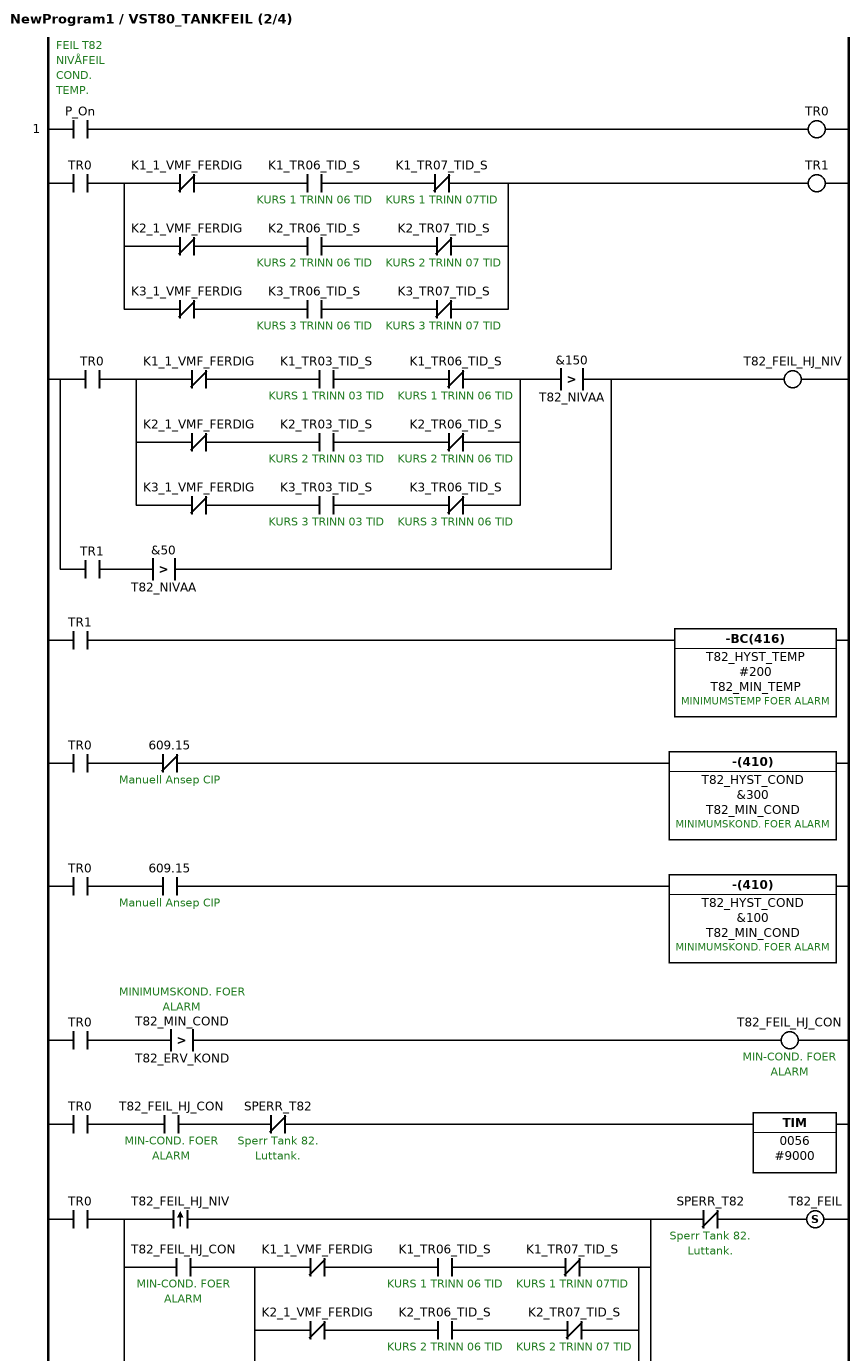

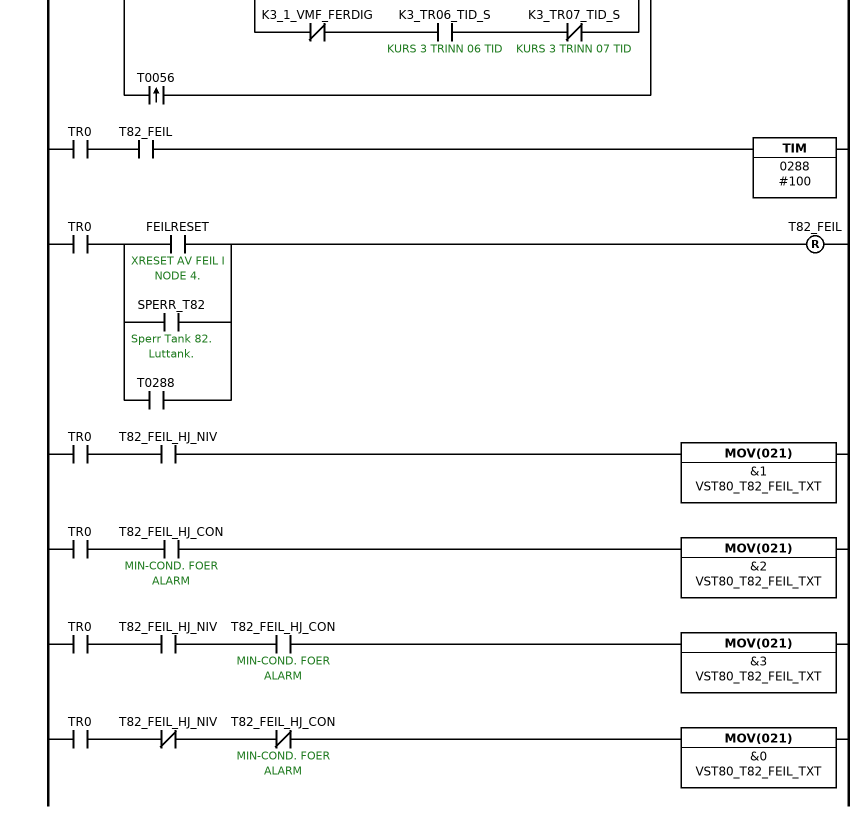
; rung 1: FEIL T82 / NIVÅFEIL / COND. / TEMP.
LD P_On
OUT TR0
LDNOT K1_1_VMF_FERDIG
AND K1_TR03_TID_S  ; KURS 1 TRINN 03 TID
ANDNOT K1_TR06_TID_S  ; KURS 1 TRINN 06 TID
LDNOT K2_1_VMF_FERDIG
AND K2_TR03_TID_S  ; KURS 2 TRINN 03 TID
ANDNOT K2_TR06_TID_S  ; KURS 2 TRINN 06 TID
ORLD
LDNOT K3_1_VMF_FERDIG
AND K3_TR03_TID_S  ; KURS 3 TRINN 03 TID
ANDNOT K3_TR06_TID_S  ; KURS 3 TRINN 06 TID
ORLD
ANDLD
AND>(320) &150 T82_NIVAA
LD TR0
LDNOT K1_1_VMF_FERDIG
AND K1_TR06_TID_S  ; KURS 1 TRINN 06 TID
ANDNOT K1_TR07_TID_S  ; KURS 1 TRINN 07TID
LDNOT K2_1_VMF_FERDIG
AND K2_TR06_TID_S  ; KURS 2 TRINN 06 TID
ANDNOT K2_TR07_TID_S  ; KURS 2 TRINN 07 TID
ORLD
LDNOT K3_1_VMF_FERDIG
AND K3_TR06_TID_S  ; KURS 3 TRINN 06 TID
ANDNOT K3_TR07_TID_S  ; KURS 3 TRINN 07 TID
ORLD
ANDLD
OUT TR1
AND>(320) &50 T82_NIVAA
ORLD
OUT T82_FEIL_HJ_NIV
LD TR1
-BC(416) T82_HYST_TEMP #200 T82_MIN_TEMP  ; MINIMUMSTEMP FOER ALARM
LD TR0
ANDNOT 609.15  ; Manuell Ansep CIP
-(410) T82_HYST_COND &300 T82_MIN_COND  ; MINIMUMSKOND. FOER ALARM
LD TR0
AND 609.15  ; Manuell Ansep CIP
-(410) T82_HYST_COND &100 T82_MIN_COND  ; MINIMUMSKOND. FOER ALARM
LD TR0
AND>(320) T82_MIN_COND T82_ERV_KOND  ; MINIMUMSKOND. FOER ALARM
OUT T82_FEIL_HJ_CON  ; MIN-COND. FOER ALARM
LD TR0
AND T82_FEIL_HJ_CON  ; MIN-COND. FOER ALARM
ANDNOT SPERR_T82  ; Sperr Tank 82. Luttank.
TIM 0056 #9000
LD TR0
@LD T82_FEIL_HJ_NIV
LD T82_FEIL_HJ_CON  ; MIN-COND. FOER ALARM
LDNOT K1_1_VMF_FERDIG
AND K1_TR06_TID_S  ; KURS 1 TRINN 06 TID
ANDNOT K1_TR07_TID_S  ; KURS 1 TRINN 07TID
LDNOT K2_1_VMF_FERDIG
AND K2_TR06_TID_S  ; KURS 2 TRINN 06 TID
ANDNOT K2_TR07_TID_S  ; KURS 2 TRINN 07 TID
ORLD
LDNOT K3_1_VMF_FERDIG
AND K3_TR06_TID_S  ; KURS 3 TRINN 06 TID
ANDNOT K3_TR07_TID_S  ; KURS 3 TRINN 07 TID
ORLD
ANDLD
ORLD
@OR T0056
ANDLD
ANDNOT SPERR_T82  ; Sperr Tank 82. Luttank.
SET T82_FEIL
LD TR0
AND T82_FEIL
TIM 0288 #100
LD TR0
LD FEILRESET  ; XRESET AV FEIL I NODE 4.
OR SPERR_T82  ; Sperr Tank 82. Luttank.
OR T0288
ANDLD
RSET T82_FEIL
LD TR0
AND T82_FEIL_HJ_NIV
MOV(021) &1 VST80_T82_FEIL_TXT
LD TR0
AND T82_FEIL_HJ_CON  ; MIN-COND. FOER ALARM
MOV(021) &2 VST80_T82_FEIL_TXT
LD TR0
AND T82_FEIL_HJ_NIV
AND T82_FEIL_HJ_CON  ; MIN-COND. FOER ALARM
MOV(021) &3 VST80_T82_FEIL_TXT
LD TR0
ANDNOT T82_FEIL_HJ_NIV
ANDNOT T82_FEIL_HJ_CON  ; MIN-COND. FOER ALARM
MOV(021) &0 VST80_T82_FEIL_TXT

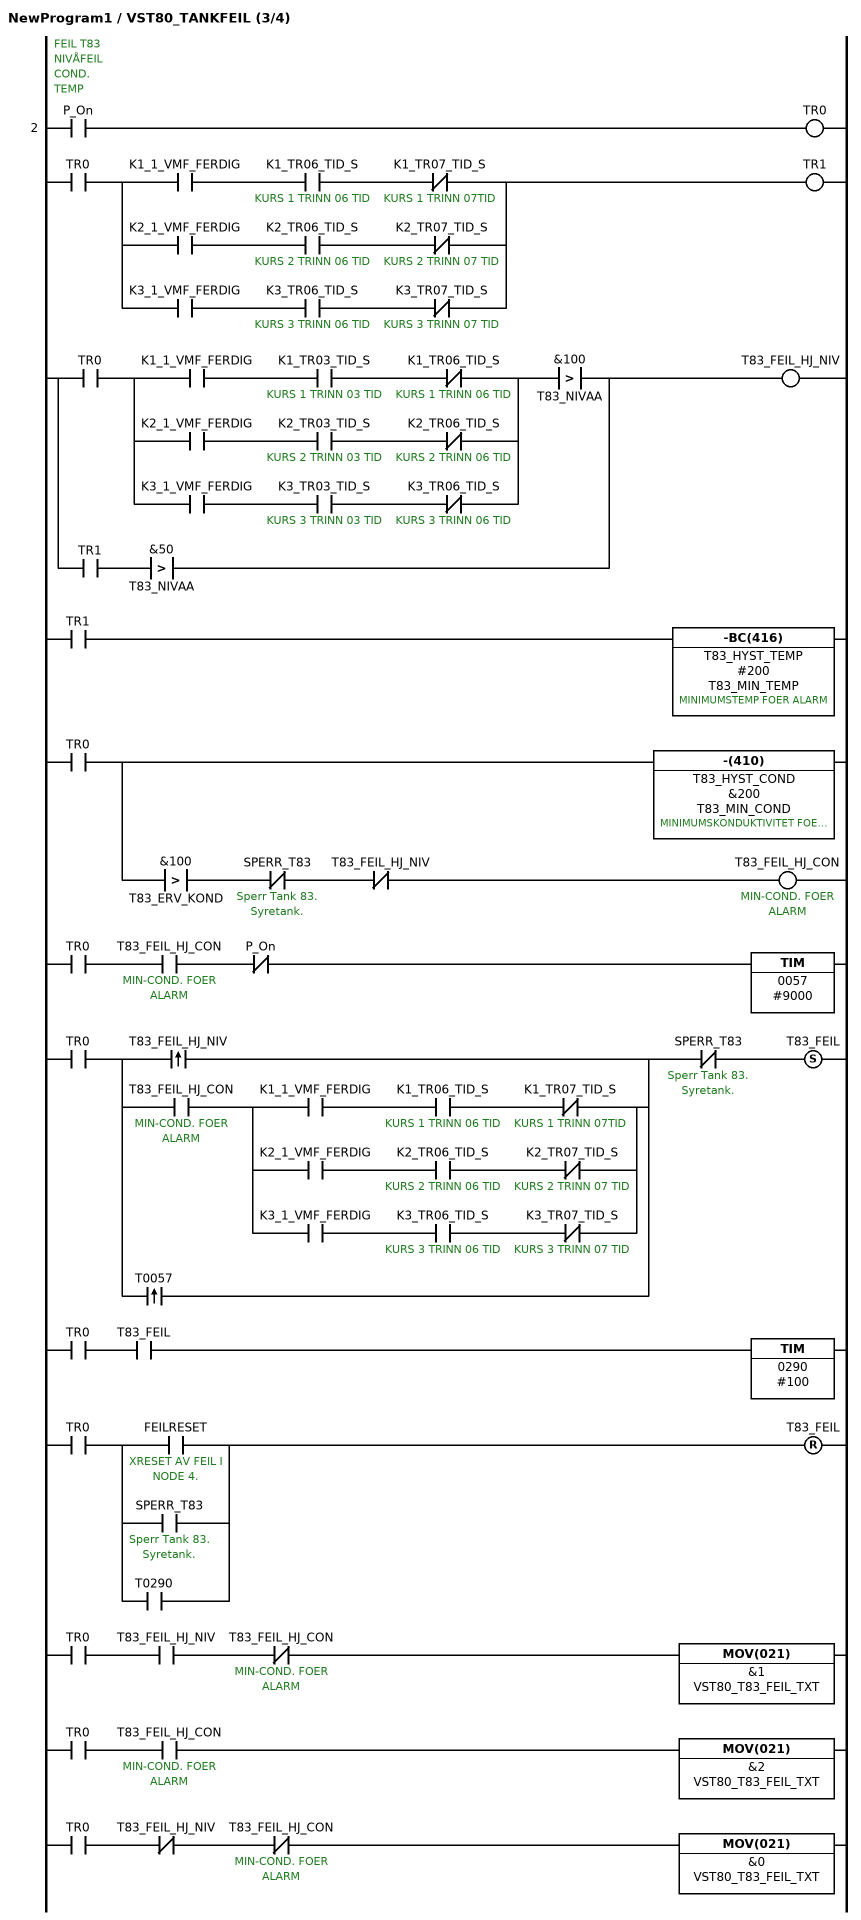
; rung 2: FEIL T83 / NIVÅFEIL / COND. / TEMP
LD P_On
OUT TR0
LD K1_1_VMF_FERDIG
AND K1_TR03_TID_S  ; KURS 1 TRINN 03 TID
ANDNOT K1_TR06_TID_S  ; KURS 1 TRINN 06 TID
LD K2_1_VMF_FERDIG
AND K2_TR03_TID_S  ; KURS 2 TRINN 03 TID
ANDNOT K2_TR06_TID_S  ; KURS 2 TRINN 06 TID
ORLD
LD K3_1_VMF_FERDIG
AND K3_TR03_TID_S  ; KURS 3 TRINN 03 TID
ANDNOT K3_TR06_TID_S  ; KURS 3 TRINN 06 TID
ORLD
ANDLD
AND>(320) &100 T83_NIVAA
LD TR0
LD K1_1_VMF_FERDIG
AND K1_TR06_TID_S  ; KURS 1 TRINN 06 TID
ANDNOT K1_TR07_TID_S  ; KURS 1 TRINN 07TID
LD K2_1_VMF_FERDIG
AND K2_TR06_TID_S  ; KURS 2 TRINN 06 TID
ANDNOT K2_TR07_TID_S  ; KURS 2 TRINN 07 TID
ORLD
LD K3_1_VMF_FERDIG
AND K3_TR06_TID_S  ; KURS 3 TRINN 06 TID
ANDNOT K3_TR07_TID_S  ; KURS 3 TRINN 07 TID
ORLD
ANDLD
OUT TR1
AND>(320) &50 T83_NIVAA
ORLD
OUT T83_FEIL_HJ_NIV
LD TR1
-BC(416) T83_HYST_TEMP #200 T83_MIN_TEMP  ; MINIMUMSTEMP FOER ALARM
LD TR0
-(410) T83_HYST_COND &200 T83_MIN_COND  ; MINIMUMSKONDUKTIVITET FOER ALARM
AND>(320) &100 T83_ERV_KOND
ANDNOT SPERR_T83  ; Sperr Tank 83. Syretank.
ANDNOT T83_FEIL_HJ_NIV
OUT T83_FEIL_HJ_CON  ; MIN-COND. FOER ALARM
LD TR0
AND T83_FEIL_HJ_CON  ; MIN-COND. FOER ALARM
ANDNOT P_On
TIM 0057 #9000
LD TR0
@LD T83_FEIL_HJ_NIV
LD T83_FEIL_HJ_CON  ; MIN-COND. FOER ALARM
LD K1_1_VMF_FERDIG
AND K1_TR06_TID_S  ; KURS 1 TRINN 06 TID
ANDNOT K1_TR07_TID_S  ; KURS 1 TRINN 07TID
LD K2_1_VMF_FERDIG
AND K2_TR06_TID_S  ; KURS 2 TRINN 06 TID
ANDNOT K2_TR07_TID_S  ; KURS 2 TRINN 07 TID
ORLD
LD K3_1_VMF_FERDIG
AND K3_TR06_TID_S  ; KURS 3 TRINN 06 TID
ANDNOT K3_TR07_TID_S  ; KURS 3 TRINN 07 TID
ORLD
ANDLD
ORLD
@OR T0057
ANDLD
ANDNOT SPERR_T83  ; Sperr Tank 83. Syretank.
SET T83_FEIL
LD TR0
AND T83_FEIL
TIM 0290 #100
LD TR0
LD FEILRESET  ; XRESET AV FEIL I NODE 4.
OR SPERR_T83  ; Sperr Tank 83. Syretank.
OR T0290
ANDLD
RSET T83_FEIL
LD TR0
AND T83_FEIL_HJ_NIV
ANDNOT T83_FEIL_HJ_CON  ; MIN-COND. FOER ALARM
MOV(021) &1 VST80_T83_FEIL_TXT
LD TR0
AND T83_FEIL_HJ_CON  ; MIN-COND. FOER ALARM
MOV(021) &2 VST80_T83_FEIL_TXT
LD TR0
ANDNOT T83_FEIL_HJ_NIV
ANDNOT T83_FEIL_HJ_CON  ; MIN-COND. FOER ALARM
MOV(021) &0 VST80_T83_FEIL_TXT

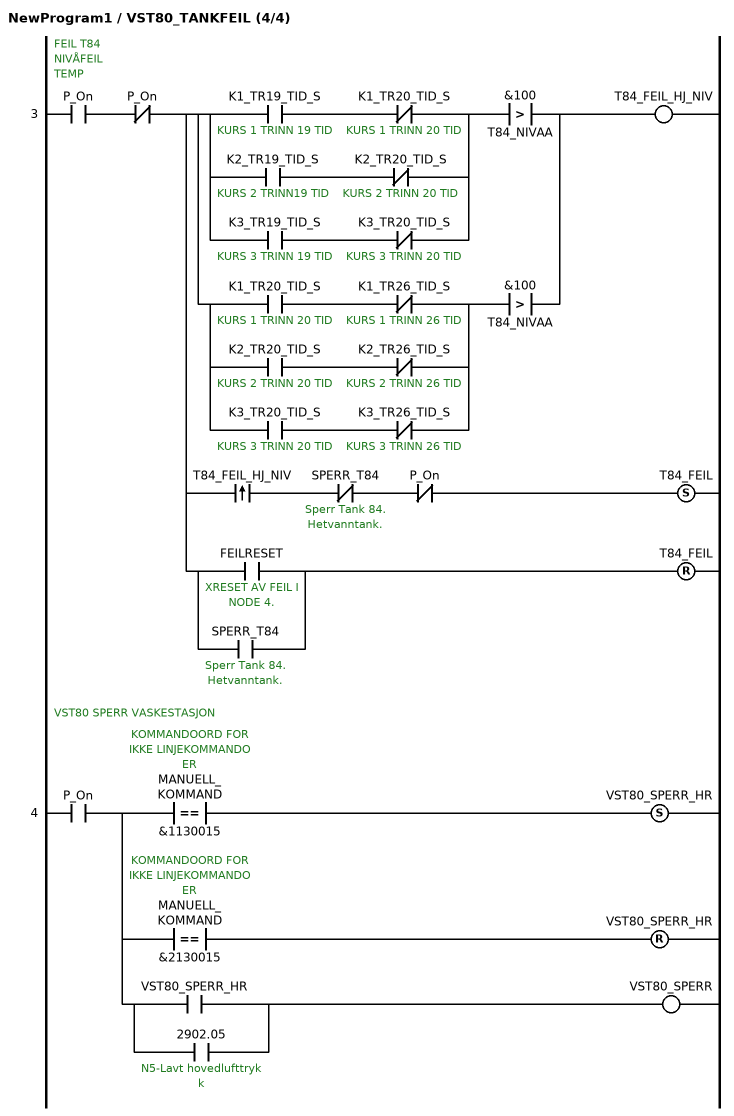
; rung 3: FEIL T84 / NIVÅFEIL / TEMP
LD P_On
ANDNOT P_On
OUT TR0
LD K1_TR19_TID_S  ; KURS 1 TRINN 19 TID
ANDNOT K1_TR20_TID_S  ; KURS 1 TRINN 20 TID
LD K2_TR19_TID_S  ; KURS 2 TRINN19 TID
ANDNOT K2_TR20_TID_S  ; KURS 2 TRINN 20 TID
ORLD
LD K3_TR19_TID_S  ; KURS 3 TRINN 19 TID
ANDNOT K3_TR20_TID_S  ; KURS 3 TRINN 20 TID
ORLD
AND>(320) &100 T84_NIVAA
LD K1_TR20_TID_S  ; KURS 1 TRINN 20 TID
ANDNOT K1_TR26_TID_S  ; KURS 1 TRINN 26 TID
LD K2_TR20_TID_S  ; KURS 2 TRINN 20 TID
ANDNOT K2_TR26_TID_S  ; KURS 2 TRINN 26 TID
ORLD
LD K3_TR20_TID_S  ; KURS 3 TRINN 20 TID
ANDNOT K3_TR26_TID_S  ; KURS 3 TRINN 26 TID
ORLD
AND>(320) &100 T84_NIVAA
ORLD
ANDLD
OUT T84_FEIL_HJ_NIV
LD TR0
@AND T84_FEIL_HJ_NIV
ANDNOT SPERR_T84  ; Sperr Tank 84. Hetvanntank.
ANDNOT P_On
SET T84_FEIL
LD TR0
LD FEILRESET  ; XRESET AV FEIL I NODE 4.
OR SPERR_T84  ; Sperr Tank 84. Hetvanntank.
ANDLD
RSET T84_FEIL
; rung 4: VST80 SPERR VASKESTASJON
LD P_On
OUT TR0
AND=L(301) MANUELL_KOMMAND &1130015  ; KOMMANDOORD FOR IKKE LINJEKOMMANDOER
SET VST80_SPERR_HR
LD TR0
AND=L(301) MANUELL_KOMMAND &2130015  ; KOMMANDOORD FOR IKKE LINJEKOMMANDOER
RSET VST80_SPERR_HR
LD TR0
LD VST80_SPERR_HR
OR 2902.05  ; N5-Lavt hovedlufttrykk
ANDLD
OUT VST80_SPERR

### Section VST80_K_1_TIDER_TR1_18

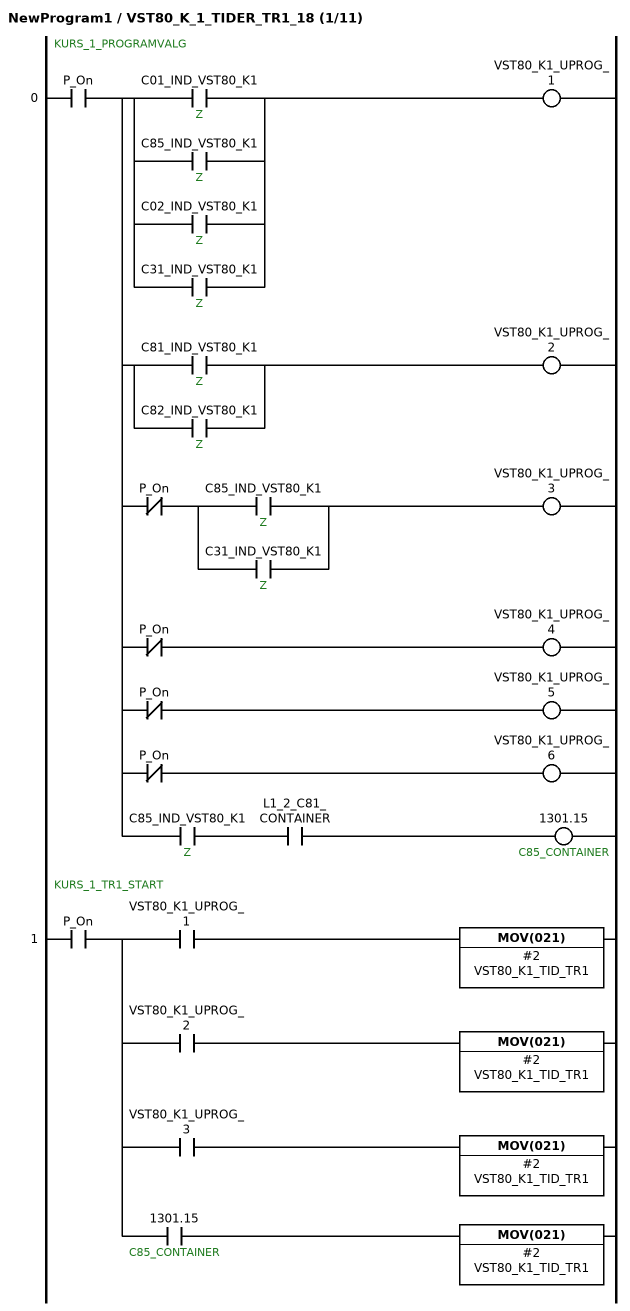
; rung 0: KURS_1_PROGRAMVALG
LD P_On
OUT TR0
LD C01_IND_VST80_K1  ; Z
OR C85_IND_VST80_K1  ; Z
OR C02_IND_VST80_K1  ; Z
OR C31_IND_VST80_K1  ; Z
ANDLD
OUT VST80_K1_UPROG_1
LD TR0
LD C81_IND_VST80_K1  ; Z
OR C82_IND_VST80_K1  ; Z
ANDLD
OUT VST80_K1_UPROG_2
LD TR0
ANDNOT P_On
LD C85_IND_VST80_K1  ; Z
OR C31_IND_VST80_K1  ; Z
ANDLD
OUT VST80_K1_UPROG_3
LD TR0
ANDNOT P_On
OUT VST80_K1_UPROG_4
LD TR0
ANDNOT P_On
OUT VST80_K1_UPROG_5
LD TR0
ANDNOT P_On
OUT VST80_K1_UPROG_6
LD TR0
AND C85_IND_VST80_K1  ; Z
AND L1_2_C81_CONTAINER
OUT 1301.15  ; C85_CONTAINER
; rung 1: KURS_1_TR1_START
LD P_On
OUT TR0
AND VST80_K1_UPROG_1
MOV(021) #2 VST80_K1_TID_TR1
LD TR0
AND VST80_K1_UPROG_2
MOV(021) #2 VST80_K1_TID_TR1
LD TR0
AND VST80_K1_UPROG_3
MOV(021) #2 VST80_K1_TID_TR1
LD TR0
AND 1301.15  ; C85_CONTAINER
MOV(021) #2 VST80_K1_TID_TR1

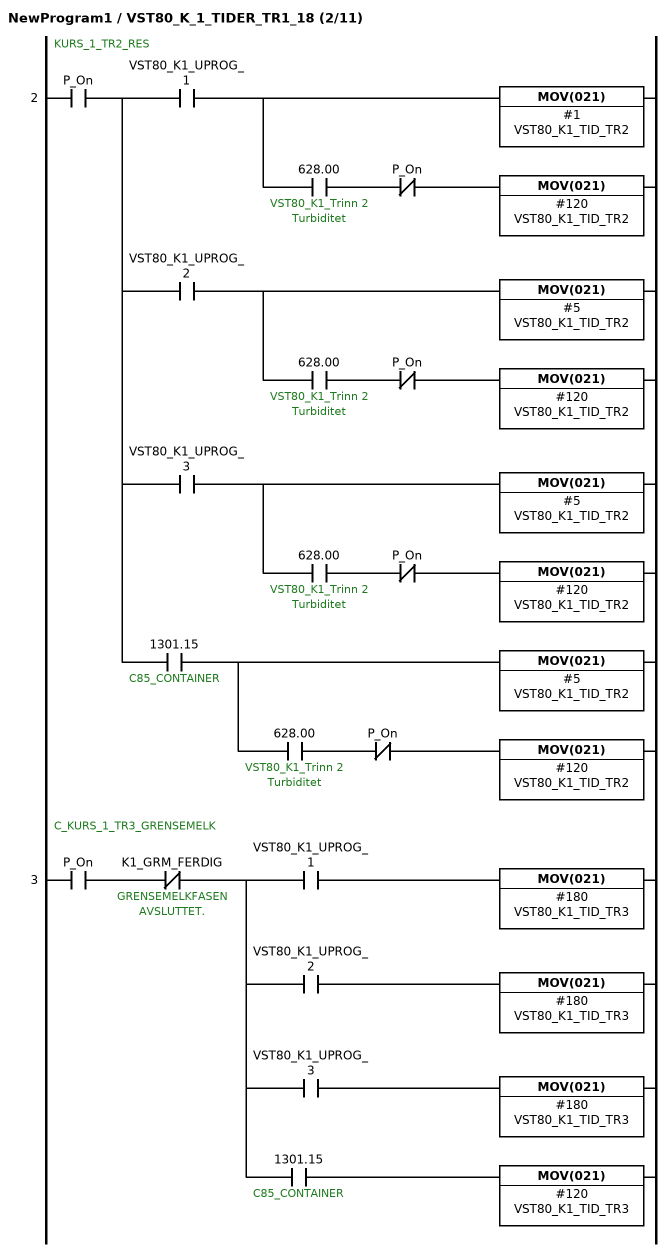
; rung 2: KURS_1_TR2_RES
LD P_On
OUT TR0
AND VST80_K1_UPROG_1
MOV(021) #1 VST80_K1_TID_TR2
AND 628.00  ; VST80_K1_Trinn 2 Turbiditet
ANDNOT P_On
MOV(021) #120 VST80_K1_TID_TR2
LD TR0
AND VST80_K1_UPROG_2
MOV(021) #5 VST80_K1_TID_TR2
AND 628.00  ; VST80_K1_Trinn 2 Turbiditet
ANDNOT P_On
MOV(021) #120 VST80_K1_TID_TR2
LD TR0
AND VST80_K1_UPROG_3
MOV(021) #5 VST80_K1_TID_TR2
AND 628.00  ; VST80_K1_Trinn 2 Turbiditet
ANDNOT P_On
MOV(021) #120 VST80_K1_TID_TR2
LD TR0
AND 1301.15  ; C85_CONTAINER
MOV(021) #5 VST80_K1_TID_TR2
AND 628.00  ; VST80_K1_Trinn 2 Turbiditet
ANDNOT P_On
MOV(021) #120 VST80_K1_TID_TR2
; rung 3: C_KURS_1_TR3_GRENSEMELK
LD P_On
ANDNOT K1_GRM_FERDIG  ; GRENSEMELKFASEN AVSLUTTET.
OUT TR0
AND VST80_K1_UPROG_1
MOV(021) #180 VST80_K1_TID_TR3
LD TR0
AND VST80_K1_UPROG_2
MOV(021) #180 VST80_K1_TID_TR3
LD TR0
AND VST80_K1_UPROG_3
MOV(021) #180 VST80_K1_TID_TR3
LD TR0
AND 1301.15  ; C85_CONTAINER
MOV(021) #120 VST80_K1_TID_TR3

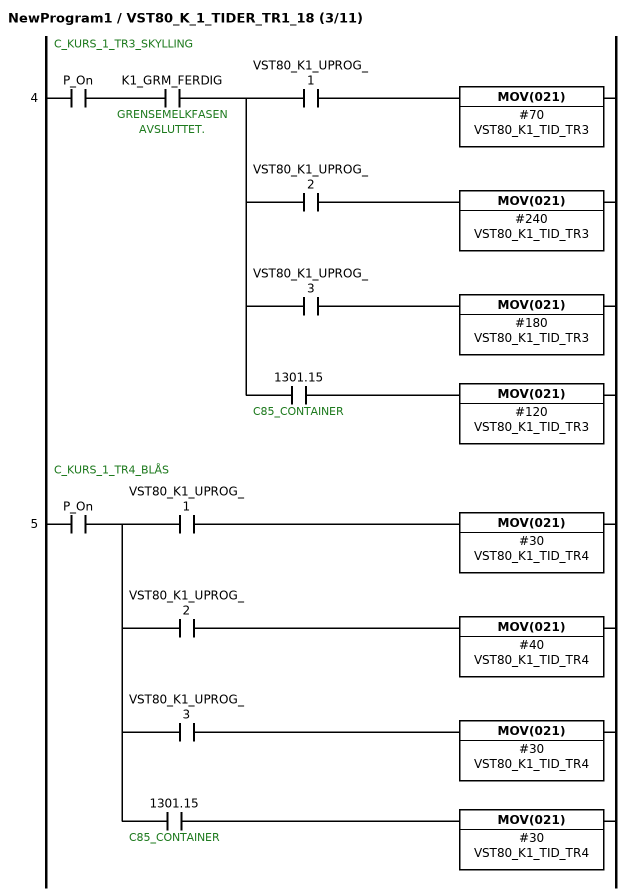
; rung 4: C_KURS_1_TR3_SKYLLING
LD P_On
AND K1_GRM_FERDIG  ; GRENSEMELKFASEN AVSLUTTET.
OUT TR0
AND VST80_K1_UPROG_1
MOV(021) #70 VST80_K1_TID_TR3
LD TR0
AND VST80_K1_UPROG_2
MOV(021) #240 VST80_K1_TID_TR3
LD TR0
AND VST80_K1_UPROG_3
MOV(021) #180 VST80_K1_TID_TR3
LD TR0
AND 1301.15  ; C85_CONTAINER
MOV(021) #120 VST80_K1_TID_TR3
; rung 5: C_KURS_1_TR4_BLÅS
LD P_On
OUT TR0
AND VST80_K1_UPROG_1
MOV(021) #30 VST80_K1_TID_TR4
LD TR0
AND VST80_K1_UPROG_2
MOV(021) #40 VST80_K1_TID_TR4
LD TR0
AND VST80_K1_UPROG_3
MOV(021) #30 VST80_K1_TID_TR4
LD TR0
AND 1301.15  ; C85_CONTAINER
MOV(021) #30 VST80_K1_TID_TR4

